PROGRAM MAIN
VAR
END_VAR

POURunLight();

END_PROGRAM

(* stored: Version 1.1.0.1, ProductVersion 3.1.4022.3
   POU MAIN: Id {225556a8-6f5f-446d-9123-a31672c626f3}, SpecialFunc None *)
